SUBAPPLICATION Uebung_072b (* GBSD auf UT ausgeben, mit Impulsen. *)
  (* Standard: 61499-2; Description: Copyright (c) 2023 Meisterschulen am Ostbahnhof This program and the accompanying materials are made available under the terms of the Eclipse Public License 2.0 which is available at https://www.eclipse.org/legal/epl-2.0/ SPDX-License-Identifier: EPL-2.0 *)
  (* Version 1.0, 2023-10-23, Franz Höpfinger, Meisterschulen am Ostbahnhof, initial API and implementation and/or initial documentation *)
  PACKAGE Uebungen;
  IMPORT Uebungen::const::UT::TECU::DefaultPool_TECU::NumberVariable_Ground_based_machine_speed;
  IMPORT Uebungen::const::UT::TECU::DefaultPool_TECU::NumberVariable_Wheel_based_machine_distance;
  IMPORT Uebungen::const::UT::TECU::DefaultPool_TECU::NumberVariable_Wheel_based_machine_speed;
  IMPORT logiBUS::io::DQ::logiBUS_DO::Output_Q1;
  IMPORT logiBUS::io::DQ::logiBUS_DO::Output_Q2;
  IMPORT logiBUS::io::DQ::logiBUS_DO::Output_Q3;
  IMPORT logiBUS::io::DQ::logiBUS_DO::Output_Q4;
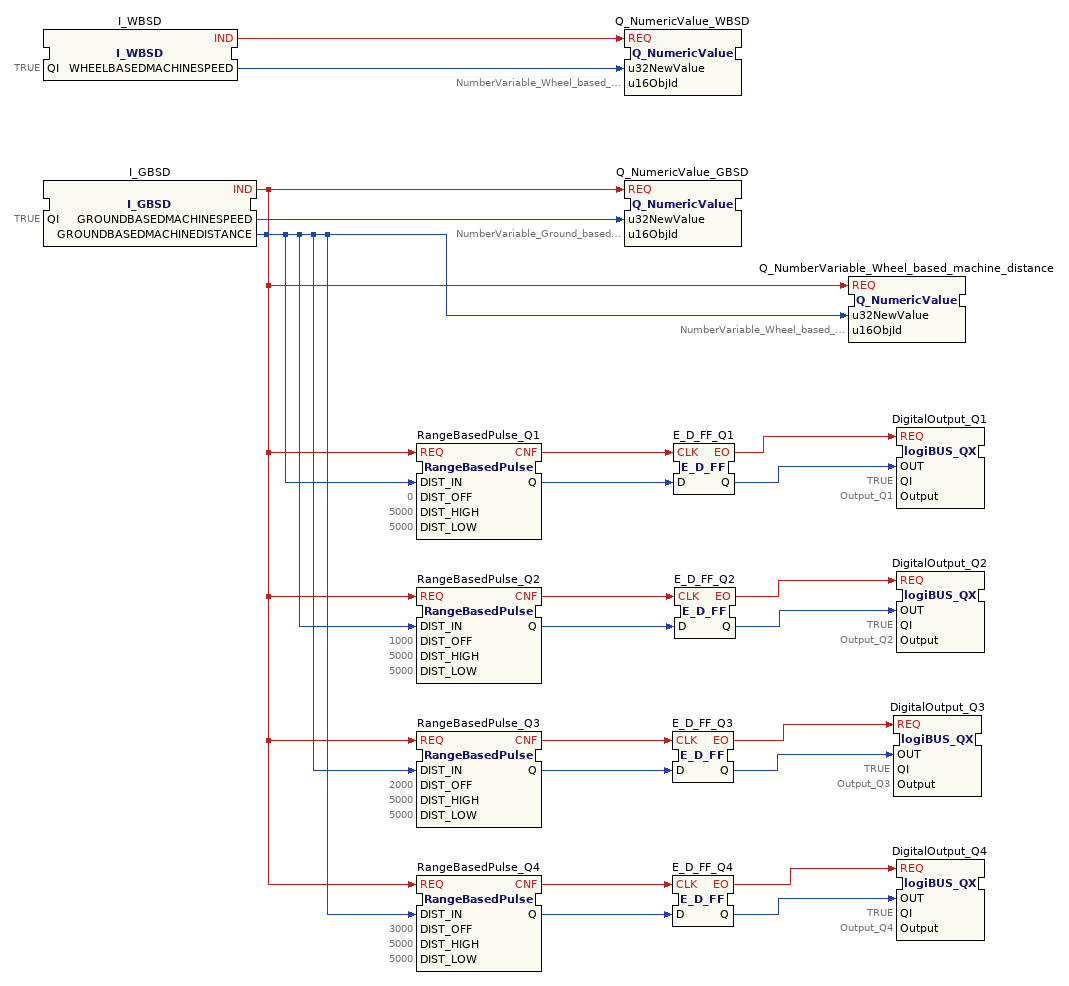
  FBS
    I_GBSD : isobus::tecu::I_GBSD(QI := TRUE);
    Q_NumericValue_GBSD : isobus::UT::Q::Q_NumericValue(u16ObjId := NumberVariable_Ground_based_machine_speed);
    I_WBSD : isobus::tecu::I_WBSD(QI := TRUE);
    Q_NumericValue_WBSD : isobus::UT::Q::Q_NumericValue(u16ObjId := NumberVariable_Wheel_based_machine_speed);
    Q_NumberVariable_Wheel_based_machine_distance : isobus::UT::Q::Q_NumericValue(u16ObjId := NumberVariable_Wheel_based_machine_distance);
    DigitalOutput_Q1 : logiBUS::io::DQ::logiBUS_QX(QI := TRUE, Output := Output_Q1);
    RangeBasedPulse_Q1 : eclipse4diac::signalprocessing::distance::RangeBasedPulse(DIST_OFF := 0, DIST_HIGH := 5000, DIST_LOW := 5000);
    E_D_FF_Q1 : iec61499::events::E_D_FF;
    DigitalOutput_Q2 : logiBUS::io::DQ::logiBUS_QX(QI := TRUE, Output := Output_Q2);
    RangeBasedPulse_Q2 : eclipse4diac::signalprocessing::distance::RangeBasedPulse(DIST_OFF := 1000, DIST_HIGH := 5000, DIST_LOW := 5000);
    E_D_FF_Q2 : iec61499::events::E_D_FF;
    DigitalOutput_Q3 : logiBUS::io::DQ::logiBUS_QX(QI := TRUE, Output := Output_Q3);
    RangeBasedPulse_Q3 : eclipse4diac::signalprocessing::distance::RangeBasedPulse(DIST_OFF := 2000, DIST_HIGH := 5000, DIST_LOW := 5000);
    E_D_FF_Q3 : iec61499::events::E_D_FF;
    DigitalOutput_Q4 : logiBUS::io::DQ::logiBUS_QX(QI := TRUE, Output := Output_Q4);
    RangeBasedPulse_Q4 : eclipse4diac::signalprocessing::distance::RangeBasedPulse(DIST_OFF := 3000, DIST_HIGH := 5000, DIST_LOW := 5000);
    E_D_FF_Q4 : iec61499::events::E_D_FF;
  END_FBS
  EVENT_CONNECTIONS
    I_GBSD.IND TO Q_NumericValue_GBSD.REQ;
    I_WBSD.IND TO Q_NumericValue_WBSD.REQ;
    E_D_FF_Q1.EO TO DigitalOutput_Q1.REQ;
    I_GBSD.IND TO Q_NumberVariable_Wheel_based_machine_distance.REQ;
    E_D_FF_Q2.EO TO DigitalOutput_Q2.REQ;
    E_D_FF_Q3.EO TO DigitalOutput_Q3.REQ;
    E_D_FF_Q4.EO TO DigitalOutput_Q4.REQ;
    I_GBSD.IND TO RangeBasedPulse_Q1.REQ;
    RangeBasedPulse_Q1.CNF TO E_D_FF_Q1.CLK;
    I_GBSD.IND TO RangeBasedPulse_Q2.REQ;
    RangeBasedPulse_Q2.CNF TO E_D_FF_Q2.CLK;
    I_GBSD.IND TO RangeBasedPulse_Q3.REQ;
    RangeBasedPulse_Q3.CNF TO E_D_FF_Q3.CLK;
    I_GBSD.IND TO RangeBasedPulse_Q4.REQ;
    RangeBasedPulse_Q4.CNF TO E_D_FF_Q4.CLK;
  END_CONNECTIONS
  DATA_CONNECTIONS
    I_GBSD.GROUNDBASEDMACHINESPEED TO Q_NumericValue_GBSD.u32NewValue;
    I_WBSD.WHEELBASEDMACHINESPEED TO Q_NumericValue_WBSD.u32NewValue;
    E_D_FF_Q1.Q TO DigitalOutput_Q1.OUT;
    I_GBSD.GROUNDBASEDMACHINEDISTANCE TO Q_NumberVariable_Wheel_based_machine_distance.u32NewValue;
    E_D_FF_Q2.Q TO DigitalOutput_Q2.OUT;
    E_D_FF_Q3.Q TO DigitalOutput_Q3.OUT;
    E_D_FF_Q4.Q TO DigitalOutput_Q4.OUT;
    I_GBSD.GROUNDBASEDMACHINEDISTANCE TO RangeBasedPulse_Q1.DIST_IN;
    RangeBasedPulse_Q1.Q TO E_D_FF_Q1.D;
    I_GBSD.GROUNDBASEDMACHINEDISTANCE TO RangeBasedPulse_Q2.DIST_IN;
    RangeBasedPulse_Q2.Q TO E_D_FF_Q2.D;
    I_GBSD.GROUNDBASEDMACHINEDISTANCE TO RangeBasedPulse_Q3.DIST_IN;
    RangeBasedPulse_Q3.Q TO E_D_FF_Q3.D;
    I_GBSD.GROUNDBASEDMACHINEDISTANCE TO RangeBasedPulse_Q4.DIST_IN;
    RangeBasedPulse_Q4.Q TO E_D_FF_Q4.D;
  END_CONNECTIONS
END_SUBAPPLICATION
